Omron CX-Programmer project NewProject (CX-Programmer 9.61)

# PLC DRILING: CP1H XA

## Global symbols (name address type ; comment)
0.00 BOOL  ; START
0.02 BOOL  ; DETECTED SENS
0.03 BOOL  ; VISION SENSOR
0.04 BOOL  ; VISION SENS
100.00 BOOL  ; CONVEYOR
100.01 BOOL  ; DRILING
100.02 BOOL  ; EMITTER
100.03 BOOL  ; PUSHER
T0000 BOOL  ; TIMER DRILLING

## Program NewProgram1 (cyclic task 0)

### Section Section1

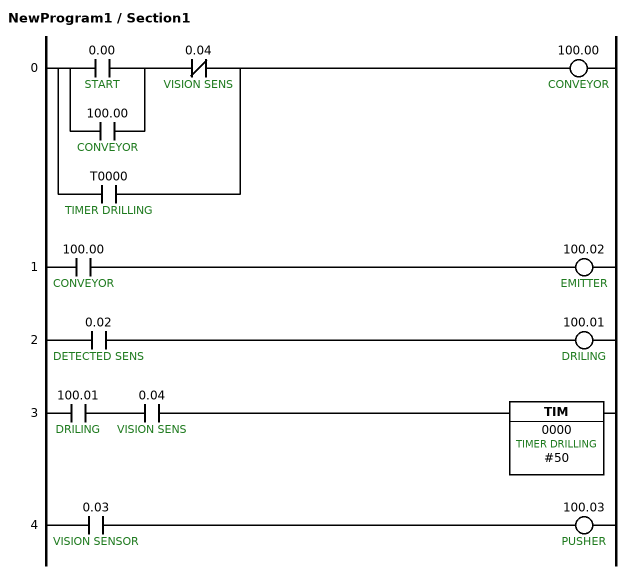
; rung 0
LD 0.00  ; START
OR 100.00  ; CONVEYOR
ANDNOT 0.04  ; VISION SENS
OR T0000  ; TIMER DRILLING
OUT 100.00  ; CONVEYOR
; rung 1
LD 100.00  ; CONVEYOR
OUT 100.02  ; EMITTER
; rung 2
LD 0.02  ; DETECTED SENS
OUT 100.01  ; DRILING
; rung 3
LD 100.01  ; DRILING
AND 0.04  ; VISION SENS
TIM 0000 #50  ; TIMER DRILLING
; rung 4
LD 0.03  ; VISION SENSOR
OUT 100.03  ; PUSHER

### Section END
; rung 0
END(001)